{attribute 'qualified_only'}
{attribute 'strict'}
TYPE E_CRYO_CTRL_CMD :
(
	NONE	:= 0,
	PRECOOL,
	COOL,
	WARM_UP,
	REPRESSURIZE
);
END_TYPE

(* stored: Version 1.1.0.1, ProductVersion 3.1.4024.9
   DUT E_CRYO_CTRL_CMD: Id {83219e50-94ed-4d54-afc2-12f1385196f1} *)
